FUNCTION_BLOCK FB_TypeShift
VAR_INPUT
	index			: INT;
	fromSt			: INT;
	toSt			: INT;
	shuttleAllowed	: BOOL;
END_VAR
VAR_OUTPUT
END_VAR
VAR
	enabled			: BOOL;
	shiftDelay		: TON;
END_VAR

//enabled := NOT typeTr[index].withPart AND NOT typeSt[toSt].withPart AND typeSt[fromSt].jobDone;
enabled :=	NOT typeSt[toSt].withPart
			AND typeSt[fromSt].withPart 
			AND typeSt[fromSt].jobDone 
			AND NOT typeSt[fromSt].hold;

shiftDelay(IN:= enabled, PT:= T#500MS);

IF shiftDelay.Q THEN
	typeSt[toSt].part	:= typeSt[fromSt].part;
	typeSt[fromSt].part	:= typeSt[0].part;
	//MEMSET(destAddr:= typeSt[1].part, fillByte:= 0, n:= 1);
	typeSt[toSt].withPart := TRUE;
	typeSt[FromSt].withPart := FALSE;	
END_IF

END_FUNCTION_BLOCK

(* stored: Version 1.1.0.1
   POU FB_TypeShift: Id {a2ab9e6d-2b63-4ebb-a471-468cf27d201c}, SpecialFunc None *)
